FUNCTION_BLOCK T_ClassThatHandlesNotifications IMPLEMENTS I_NotificationHandler
VAR_INPUT
END_VAR
VAR_OUTPUT
END_VAR
VAR
    _NotificationCount : UDINT;
    _Identifier : STRING;
END_VAR

PROPERTY NotificationCallCount : UDINT
GET
NotificationCallCount := _NotificationCount;
END_GET
END_PROPERTY

METHOD OnNotificationReceived
VAR_INPUT
    NotificationId   : UDINT;
    NotificationName : T_MaxString;
    Args             : IStreamReader;
END_VAR
IF NotificationId = E_Test_NotificationId.OnPbPressed_Notification THEN 
    // Notification Id maps to Handler method name here...
    
    OnPbPressed(Identifier := Args.Read_STRING());   
END_IF
END_METHOD

METHOD OnPbPressed
VAR_INPUT
    Identifier : STRING;
END_VAR
_Identifier := Identifier;
_NotificationCount := _NotificationCount + 1;
END_METHOD

END_FUNCTION_BLOCK

(* stored: Version 1.1.0.1, ProductVersion 3.1.4024.5
   POU T_ClassThatHandlesNotifications: Id {86eb1b79-63f5-4257-8b9b-6105f01b6690}, SpecialFunc None
   Property NotificationCallCount: Id {e2095a8f-63c5-46d0-9bbf-aaec0fa11803}
   Get Get: Id {31441469-2fb2-4415-8f79-e88239624682}
   Method OnNotificationReceived: Id {d81e77bc-ceca-4b34-b455-87073507d115}
   Method OnPbPressed: Id {630a0f00-37f3-4161-a052-3351be3ac105} *)
